# EPICS autosave request: delaygenApp/Db/drvDG645_settings.req
$(P)$(R)Label

$(P)$(R)T0OutputAmpTweakAO
$(P)$(R)ABOutputAmpTweakAO
$(P)$(R)CDOutputAmpTweakAO
$(P)$(R)EFOutputAmpTweakAO
$(P)$(R)GHOutputAmpTweakAO

$(P)$(R)T0OutputOffsetTweakAO
$(P)$(R)ABOutputOffsetTweakAO
$(P)$(R)CDOutputOffsetTweakAO
$(P)$(R)EFOutputOffsetTweakAO
$(P)$(R)GHOutputOffsetTweakAO
